// TIA Portal V16 export
// export: Created 2024-12-03T15:41:45.5032102Z, ExportSetting WithReadOnly, DisplayName Totally Integrated Automation Portal, DisplayVersion V16 Update 6, DisplayName TIA Portal Version Control Interface, DisplayVersion V16 Update 2, DisplayName TIA Portal Openness, DisplayVersion V16 Update 6, DisplayName TIA Portal Teamcenter Gateway, DisplayVersion V16, DisplayName SINAMICS Startdrive Advanced, DisplayVersion V16 Update 5, DisplayName SINAMICS Startdrive G130, G150, S120, S150, SINAMICS MV, S210, DisplayVersion V16 Update 5, DisplayName SINAMICS Startdrive G110M, G120, G120C, G120D, G120P, G115D, DisplayVersion V16 Update 5, DisplayName STEP 7 Professional, DisplayVersion V16 Update 6, DisplayName STEP 7 Safety, DisplayVersion V16, DisplayName WinCC Advanced / Unified PC, DisplayVersion V16 Update 6
TYPE "CONFIG_EPOS_UDT"
// stored: CreationDate 2022-02-10T10:30:20.6863124Z, InterfaceModifiedDate 2021-08-30T09:48:11.3473082Z, IsConsistent true, LibraryConformanceStatus The object is library-conformant., ModifiedDate 2021-08-30T09:48:30.4016332Z
   STRUCT
      Off2_NoPulseDisable : Bool;
      Off3_NoRampStop : Bool;
      SoftwareLimitActive : Bool;
      Stopcams : Bool;
      MeasuringInputEdgeEvaluation : Bool;
      MeasuringInputSelection : Bool;
      SignalSourceReferenceMask : Bool;
      ExternalBlockChange : Bool;
      ContinousSetPointAcceptance : Bool;
      DDS0 : Bool;
      DDS1 : Bool;
      DDS2 : Bool;
      DDS3 : Bool;
      DDS4 : Bool;
      ParkingAxisSelection : Bool;
      spare : Bool;
      spare_1 : Word;
   END_STRUCT;
END_TYPE
